(* IEC 61131-3 sources: sF/Sf/src/typeLib/modules/STBlocks, 1 file *)

(* ---- sqrtST.ST ---- *)
PROGRAM execute
VAR
    input1: REAL;
    output1: REAL;
END_VAR

output1 := input1 * input1;
END_PROGRAM
